// TIA Portal project "color based pick and place" (V16)
// Vorlageprojekt für das Buch mit Zielsystem S7-1200

(* hardware
DEVICE "S7-1200-Station_1"  S7-1200 Station
   slot 0: "Baugruppenträger_0"  Rack  V1.0
   slot 1: "PLC_1"  CPU 1211C DC/DC/DC  6ES7 211-1AE40-0XB0  V4.1
*)

// ===== PLC "PLC_1"  CPU 1211C DC/DC/DC =====

VAR_GLOBAL   // PLC tag table "Standard-Variablentabelle"
   "start" AT %I0.0 : Bool;
   "diffus1" AT %I0.1 : Bool;
   "vision sens" AT %I0.2 : Bool;
   "diffus2" AT %I0.3 : Bool;
   "diffuse3" AT %I0.4 : Bool;
   "emitt1" AT %Q0.0 : Bool;
   "emitt2" AT %Q0.1 : Bool;
   "emitt3" AT %Q0.2 : Bool;
   "conv1" AT %Q0.3 : Bool;
   "conv2" AT %Q0.4 : Bool;
   "conv3" AT %Q0.5 : Bool;
   "diffues2 memory" AT %M0.3 : Bool;
   "diffues3 memory" AT %M0.4 : Bool;
   "diffues1 memory" AT %M0.1 : Bool;
   "vision sensor memory" AT %M0.2 : Bool;
   "z down" AT %Q0.6 : Bool;
   "z sensor(1)" AT %I0.7 : Bool;
   "z snsor  memory" AT %M50.7 : Bool;
   "box detect(1)" AT %I1.0 : Bool;
   "box detect memo" AT %M16.0 : Bool;
   "grab" AT %Q0.7 : Bool;
   "x move" AT %Q1.0 : Bool;
   "x move sens" AT %I1.1 : Bool;
   "x sens mem" AT %M16.1 : Bool;
   "turn left" AT %Q1.1 : Bool;
   "turn right" AT %Q1.2 : Bool;
   "turn sensor" AT %I1.2 : Bool;
   "ton set" AT %M0.5 : Bool;
   "arrive" AT %M0.6 : Bool;
   "retrain" AT %M16.2 : Bool;
   "Tag_1" AT %M16.3 : Bool;
   "Tag_2" AT %M3.0 : Bool;
   "Tag_3" AT %M3.1 : Bool;
   "Tag_4" AT %M3.2 : Bool;
   "reset" AT %M120.0 : Bool;
   "counter reset" AT %I1.3 : Bool;
   "warning light" AT %Q1.3 : Bool;
   "Tag_5" AT %M3.4 : Bool;
   "Tag_6" AT %M10.0 : Bool;
   "Tag_7" AT %M10.1 : Bool;
   "Tag_8" AT %M10.4 : Bool;
   "System_Byte" AT %MB1 : Byte;
   "FirstScan" AT %M1.0 : Bool;
   "DiagStatusUpdate" AT %M1.1 : Bool;
   "AlwaysTRUE" AT %M1.2 : Bool;
   "AlwaysFALSE" AT %M1.3 : Bool;
   "Clock_Byte" AT %MB15 : Byte;
   "Clock_10Hz" AT %M15.0 : Bool;
   "Clock_5Hz" AT %M15.1 : Bool;
   "Clock_2.5Hz" AT %M15.2 : Bool;
   "Clock_2Hz" AT %M15.3 : Bool;
   "Clock_1.25Hz" AT %M15.4 : Bool;
   "Clock_1Hz" AT %M15.5 : Bool;
   "Clock_0.625Hz" AT %M15.6 : Bool;
   "Clock_0.5Hz" AT %M15.7 : Bool;
   "Tag_9" AT %M10.7 : Bool;
   "Tag_10" AT %M50.0 : Bool;
   "Tag_11" AT %M10.2 : Bool;
   "Tag_12" AT %M50.5 : Bool;
   "color not detect latch" AT %M60.0 : Bool;
   "color detect latch" AT %M60.1 : Bool;
   "Tag_13" AT %M70.0 : Bool;
   "turn right reset" AT %M90.0 : Bool;
   "Tag_14" AT %M60.6 : Bool;
   "Tag_15" AT %M100.0 : Bool;
   "Tag_16" AT %M100.1 : Bool;
   "Tag_17" AT %M600.0 : Bool;
   "Tag_18" AT %M600.1 : Bool;
   "Tag_19" AT %M300.3 : Bool;
   "Tag_20" AT %M300.4 : Bool;
   "Tag_21" AT %M700.0 : Bool;
   "Tag_22" AT %M700.1 : Bool;
END_VAR

// folder: System blocks/Program resources

DATA_BLOCK "IEC_Timer_0_DB"   // DB1
{ S7_Optimized_Access := 'TRUE' }
AUTHOR : Simatic
FAMILY : IEC
NAME : IEC_TMR
VERSION : 1.0
// stored: InstanceOfName IEC_TIMER
"IEC_TIMER"
BEGIN
END_DATA_BLOCK

DATA_BLOCK "IEC_Timer_0_DB_1"   // DB2
{ S7_Optimized_Access := 'TRUE' }
AUTHOR : Simatic
FAMILY : IEC
NAME : IEC_TMR
VERSION : 1.0
// stored: InstanceOfName IEC_TIMER
"IEC_TIMER"
BEGIN
END_DATA_BLOCK

DATA_BLOCK "IEC_Counter_0_DB"   // DB3
{ S7_Optimized_Access := 'TRUE' }
AUTHOR : Simatic
FAMILY : IEC
NAME : CNTR
VERSION : 1.0
// stored: InstanceOfName IEC_COUNTER
"IEC_COUNTER"
BEGIN
END_DATA_BLOCK

DATA_BLOCK "IEC_Timer_0_DB_3"   // DB4
{ S7_Optimized_Access := 'TRUE' }
AUTHOR : Simatic
FAMILY : IEC
NAME : IEC_TMR
VERSION : 1.0
// stored: InstanceOfName IEC_TIMER
"IEC_TIMER"
BEGIN
END_DATA_BLOCK

DATA_BLOCK "IEC_Timer_0_DB_2"   // DB5
{ S7_Optimized_Access := 'TRUE' }
AUTHOR : Simatic
FAMILY : IEC
NAME : IEC_TMR
VERSION : 1.0
// stored: InstanceOfName IEC_TIMER
"IEC_TIMER"
BEGIN
END_DATA_BLOCK

DATA_BLOCK "IEC_Counter_1_DB"   // DB6
{ S7_Optimized_Access := 'TRUE' }
AUTHOR : Simatic
FAMILY : IEC
NAME : CNTR
VERSION : 1.0
// stored: InstanceOfName IEC_COUNTER
"IEC_COUNTER"
BEGIN
END_DATA_BLOCK

DATA_BLOCK "IEC_Timer_0_DB_4"   // DB7
{ S7_Optimized_Access := 'TRUE' }
AUTHOR : Simatic
FAMILY : IEC
NAME : IEC_TMR
VERSION : 1.0
// stored: InstanceOfName IEC_TIMER
"IEC_TIMER"
BEGIN
END_DATA_BLOCK

DATA_BLOCK "IEC_Timer_0_DB_5"   // DB8
{ S7_Optimized_Access := 'TRUE' }
AUTHOR : Simatic
FAMILY : IEC
NAME : IEC_TMR
VERSION : 1.0
// stored: InstanceOfName IEC_TIMER
"IEC_TIMER"
BEGIN
END_DATA_BLOCK

// folder: (top level)

FUNCTION "color detect" : Void   // FC1, LAD
{ S7_Optimized_Access := 'TRUE' }
VERSION : 0.1
   VAR_TEMP   // added for the SCL form of the ladder/FBD networks
      _w1 : Bool;
      _w2 : Bool;
      _w3 : Bool;
   END_VAR
BEGIN

REGION Network 1
   // color detect
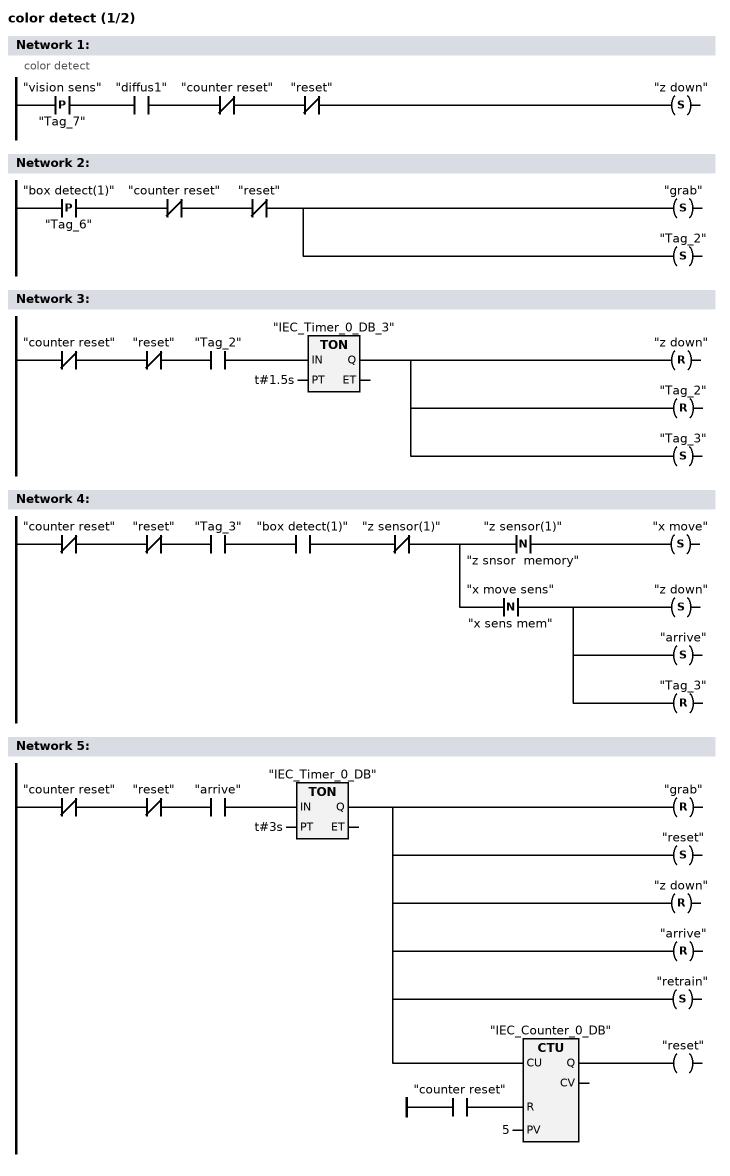
   RUNG wire#powerrail
      P_Contact(operand := "vision sens", bit := "Tag_7")
      Contact( "diffus1" )
      I_Contact( "counter reset" )
      I_Contact( "reset" )
      S_Coil( "z down" )
   END_RUNG
   // the same network as SCL:
   #_w1 := "vision sens" AND NOT "Tag_7";   // rising edge of "vision sens"
   "Tag_7" := "vision sens";
   IF #_w1 AND "diffus1" AND NOT "counter reset" AND NOT "reset" THEN "z down" := TRUE; END_IF;
END_REGION

REGION Network 2
   RUNG wire#powerrail
      P_Contact(operand := "box detect(1)", bit := "Tag_6")
      I_Contact( "counter reset" )
      I_Contact( "reset" )
      wire#w1
      S_Coil( "grab" )
   END_RUNG
   RUNG wire#w1
      S_Coil( "Tag_2" )
   END_RUNG
   // the same network as SCL:
   #_w1 := "box detect(1)" AND NOT "Tag_6";   // rising edge of "box detect(1)"
   "Tag_6" := "box detect(1)";
   IF #_w1 AND NOT "counter reset" AND NOT "reset" THEN
       "grab" := TRUE;
       "Tag_2" := TRUE;
   END_IF;
END_REGION

REGION Network 3
   "IEC_Timer_0_DB_3".TON(IN := NOT "counter reset" AND NOT "reset" AND "Tag_2", PT := t#1.5s);
   IF "IEC_Timer_0_DB_3".Q THEN
       "z down" := FALSE;
       "Tag_2" := FALSE;
       "Tag_3" := TRUE;
   END_IF;
END_REGION

REGION Network 4
   RUNG wire#powerrail
      I_Contact( "counter reset" )
      I_Contact( "reset" )
      Contact( "Tag_3" )
      Contact( "box detect(1)" )
      I_Contact( "z sensor(1)" )
      wire#w1
      N_Contact(operand := "z sensor(1)", bit := "z snsor  memory")
      S_Coil( "x move" )
   END_RUNG
   RUNG wire#w1
      N_Contact(operand := "x move sens", bit := "x sens mem")
      wire#w2
      S_Coil( "z down" )
   END_RUNG
   RUNG wire#w2
      S_Coil( "arrive" )
   END_RUNG
   RUNG wire#w2
      R_Coil( "Tag_3" )
   END_RUNG
   // the same network as SCL:
   #_w1 := NOT "counter reset" AND NOT "reset" AND "Tag_3" AND "box detect(1)" AND NOT "z sensor(1)";
   #_w2 := #_w1 AND NOT "z sensor(1)" AND "z snsor  memory";   // falling edge of "z sensor(1)"
   "z snsor  memory" := "z sensor(1)";
   IF #_w2 THEN "x move" := TRUE; END_IF;
   #_w3 := #_w1 AND NOT "x move sens" AND "x sens mem";   // falling edge of "x move sens"
   "x sens mem" := "x move sens";
   IF #_w3 THEN
       "z down" := TRUE;
       "arrive" := TRUE;
       "Tag_3" := FALSE;
   END_IF;
END_REGION

REGION Network 5
   "IEC_Timer_0_DB".TON(IN := NOT "counter reset" AND NOT "reset" AND "arrive", PT := t#3s);
   IF "IEC_Timer_0_DB".Q THEN
       "grab" := FALSE;
       "reset" := TRUE;
       "z down" := FALSE;
       "arrive" := FALSE;
       "retrain" := TRUE;
   END_IF;
   "IEC_Counter_0_DB".CTU(CU := "IEC_Timer_0_DB".Q, R := "counter reset", PV := 5);
   "reset" := "IEC_Counter_0_DB".Q;
END_REGION

REGION Network 6
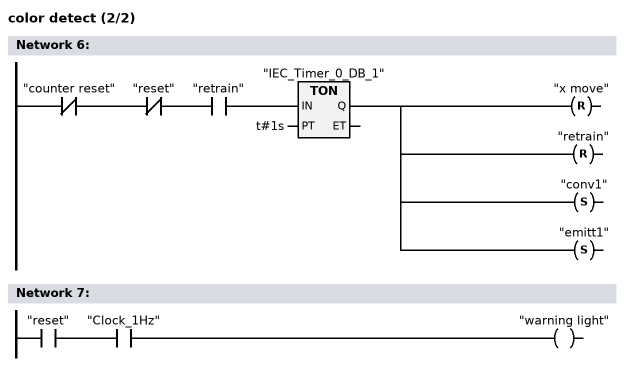
   "IEC_Timer_0_DB_1".TON(IN := NOT "counter reset" AND NOT "reset" AND "retrain", PT := t#1s);
   IF "IEC_Timer_0_DB_1".Q THEN
       "x move" := FALSE;
       "retrain" := FALSE;
       "conv1" := TRUE;
       "emitt1" := TRUE;
   END_IF;
END_REGION

REGION Network 7
   RUNG wire#powerrail
      Contact( "reset" )
      Contact( "Clock_1Hz" )
      Coil( "warning light" )
   END_RUNG
   // the same network as SCL:
   "warning light" := "reset" AND "Clock_1Hz";
END_REGION
END_FUNCTION

FUNCTION "color not detect" : Void   // FC2, LAD
{ S7_Optimized_Access := 'TRUE' }
VERSION : 0.1
   VAR_TEMP   // added for the SCL form of the ladder/FBD networks
      _w1 : Bool;
      _w2 : Bool;
      _w3 : Bool;
      _w4 : Bool;
   END_VAR
BEGIN

REGION Network 1
   // color detect
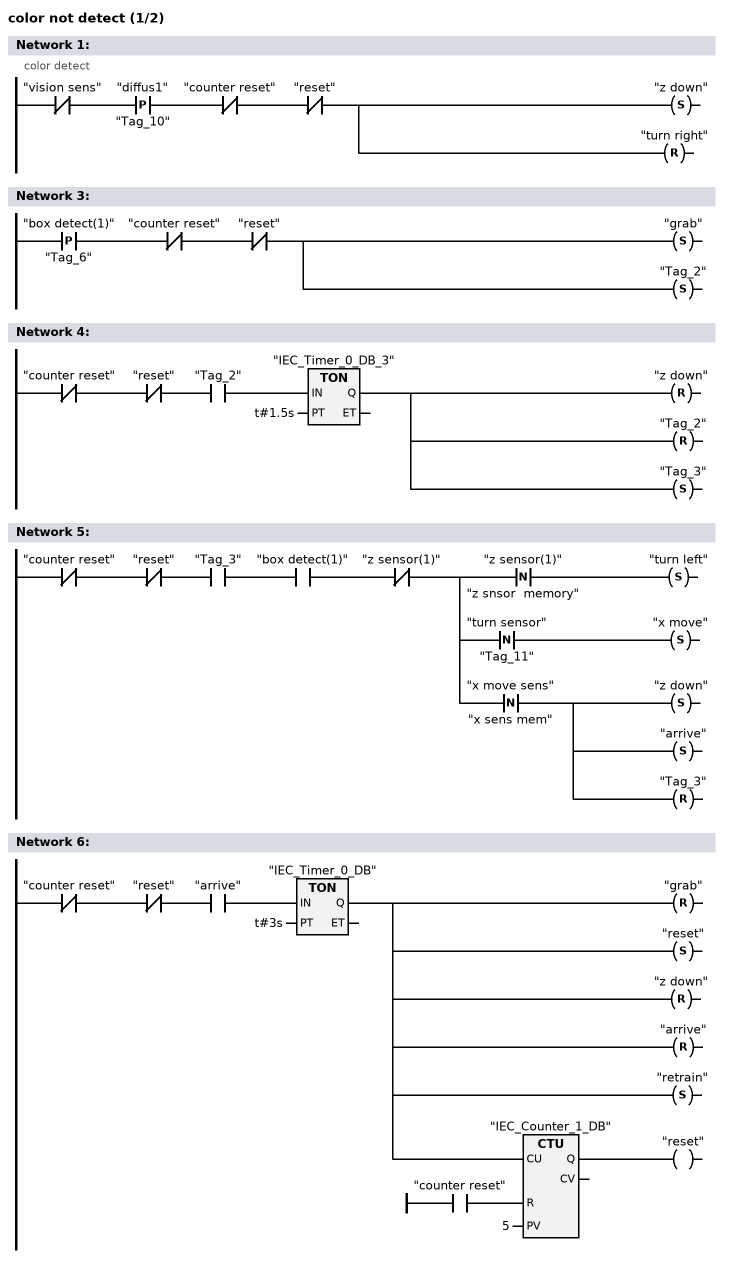
   RUNG wire#powerrail
      I_Contact( "vision sens" )
      P_Contact(operand := "diffus1", bit := "Tag_10")
      I_Contact( "counter reset" )
      I_Contact( "reset" )
      wire#w1
      S_Coil( "z down" )
   END_RUNG
   RUNG wire#w1
      R_Coil( "turn right" )
   END_RUNG
   // the same network as SCL:
   #_w1 := NOT "vision sens" AND "diffus1" AND NOT "Tag_10";   // rising edge of "diffus1"
   "Tag_10" := "diffus1";
   IF #_w1 AND NOT "counter reset" AND NOT "reset" THEN
       "z down" := TRUE;
       "turn right" := FALSE;
   END_IF;
END_REGION

REGION Network 3
   RUNG wire#powerrail
      P_Contact(operand := "box detect(1)", bit := "Tag_6")
      I_Contact( "counter reset" )
      I_Contact( "reset" )
      wire#w1
      S_Coil( "grab" )
   END_RUNG
   RUNG wire#w1
      S_Coil( "Tag_2" )
   END_RUNG
   // the same network as SCL:
   #_w1 := "box detect(1)" AND NOT "Tag_6";   // rising edge of "box detect(1)"
   "Tag_6" := "box detect(1)";
   IF #_w1 AND NOT "counter reset" AND NOT "reset" THEN
       "grab" := TRUE;
       "Tag_2" := TRUE;
   END_IF;
END_REGION

REGION Network 4
   "IEC_Timer_0_DB_3".TON(IN := NOT "counter reset" AND NOT "reset" AND "Tag_2", PT := t#1.5s);
   IF "IEC_Timer_0_DB_3".Q THEN
       "z down" := FALSE;
       "Tag_2" := FALSE;
       "Tag_3" := TRUE;
   END_IF;
END_REGION

REGION Network 5
   RUNG wire#powerrail
      I_Contact( "counter reset" )
      I_Contact( "reset" )
      Contact( "Tag_3" )
      Contact( "box detect(1)" )
      I_Contact( "z sensor(1)" )
      wire#w1
      N_Contact(operand := "z sensor(1)", bit := "z snsor  memory")
      S_Coil( "turn left" )
   END_RUNG
   RUNG wire#w1
      N_Contact(operand := "turn sensor", bit := "Tag_11")
      S_Coil( "x move" )
   END_RUNG
   RUNG wire#w1
      N_Contact(operand := "x move sens", bit := "x sens mem")
      wire#w2
      S_Coil( "z down" )
   END_RUNG
   RUNG wire#w2
      S_Coil( "arrive" )
   END_RUNG
   RUNG wire#w2
      R_Coil( "Tag_3" )
   END_RUNG
   // the same network as SCL:
   #_w1 := NOT "counter reset" AND NOT "reset" AND "Tag_3" AND "box detect(1)" AND NOT "z sensor(1)";
   #_w2 := #_w1 AND NOT "z sensor(1)" AND "z snsor  memory";   // falling edge of "z sensor(1)"
   "z snsor  memory" := "z sensor(1)";
   IF #_w2 THEN "turn left" := TRUE; END_IF;
   #_w3 := #_w1 AND NOT "turn sensor" AND "Tag_11";   // falling edge of "turn sensor"
   "Tag_11" := "turn sensor";
   IF #_w3 THEN "x move" := TRUE; END_IF;
   #_w4 := #_w1 AND NOT "x move sens" AND "x sens mem";   // falling edge of "x move sens"
   "x sens mem" := "x move sens";
   IF #_w4 THEN
       "z down" := TRUE;
       "arrive" := TRUE;
       "Tag_3" := FALSE;
   END_IF;
END_REGION

REGION Network 6
   "IEC_Timer_0_DB".TON(IN := NOT "counter reset" AND NOT "reset" AND "arrive", PT := t#3s);
   IF "IEC_Timer_0_DB".Q THEN
       "grab" := FALSE;
       "reset" := TRUE;
       "z down" := FALSE;
       "arrive" := FALSE;
       "retrain" := TRUE;
   END_IF;
   "IEC_Counter_1_DB".CTU(CU := "IEC_Timer_0_DB".Q, R := "counter reset", PV := 5);
   "reset" := "IEC_Counter_1_DB".Q;
END_REGION

REGION Network 7
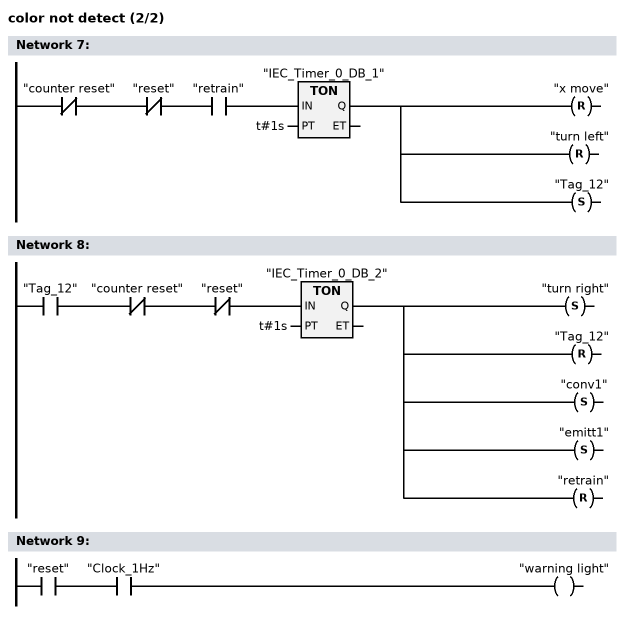
   "IEC_Timer_0_DB_1".TON(IN := NOT "counter reset" AND NOT "reset" AND "retrain", PT := t#1s);
   IF "IEC_Timer_0_DB_1".Q THEN
       "x move" := FALSE;
       "turn left" := FALSE;
       "Tag_12" := TRUE;
   END_IF;
END_REGION

REGION Network 8
   "IEC_Timer_0_DB_2".TON(IN := "Tag_12" AND NOT "counter reset" AND NOT "reset", PT := t#1s);
   IF "IEC_Timer_0_DB_2".Q THEN
       "turn right" := TRUE;
       "Tag_12" := FALSE;
       "conv1" := TRUE;
       "emitt1" := TRUE;
       "retrain" := FALSE;
   END_IF;
END_REGION

REGION Network 9
   RUNG wire#powerrail
      Contact( "reset" )
      Contact( "Clock_1Hz" )
      Coil( "warning light" )
   END_RUNG
   // the same network as SCL:
   "warning light" := "reset" AND "Clock_1Hz";
END_REGION
END_FUNCTION

FUNCTION "MHJ-PLC-Lab-Function-S71200" : Void   // FC9000, SCL
{ S7_Optimized_Access := 'TRUE' }
VERSION : 0.1
   VAR_TEMP
      rdTimeReturn : Int;
      outputTime : DTL;
      SyncVal : Byte;
      forVal : Int;
      forVal_2 : Int;
      Value : Byte;
   END_VAR
   VAR CONSTANT
      CompVal : Byte := 16#34;
      Value_01 : Byte := 16#11;
      Value_01_DW : DWord := 16#A165_D992;
      Value_02_DW : DWord := 16#58BE_4401;
   END_VAR
BEGIN

   #Value:=PEEK(area := 16#82,
        dbNumber := 0,
        byteOffset := 511);
   #Value := #Value + 1;

   POKE(area := 16#82,
        dbNumber := 0,
        byteOffset := 511,
        value := #Value);

   POKE(area:=16#81,
        dbNumber:=0,
        byteOffset:=1016,
        value:=#Value_01_DW);
   POKE(area := 16#81,
        dbNumber := 0,
        byteOffset := 1020,
        value := #Value_02_DW);

   POKE(area := 16#81,
        dbNumber := 0,
        byteOffset := 511,
        value := B#16#00);

   FOR #forVal := 0 TO 120 DO
       FOR #forVal_2:=0 TO 10 DO
           #rdTimeReturn:=RD_SYS_T(#outputTime);
           #rdTimeReturn := WR_SYS_T(#outputTime);
           #rdTimeReturn := RD_SYS_T(#outputTime);
           #rdTimeReturn := WR_SYS_T(#outputTime);
       END_FOR;
       #SyncVal:= PEEK(area := 16#81,
                      dbNumber := 0,
                      byteOffset := 511);
       IF #SyncVal = #CompVal THEN
          GOTO M_1;
       END_IF;
   END_FOR;
   RETURN;

   M_1:
   POKE(area := 16#81,
        dbNumber := 0,
        byteOffset := 511,
        value := B#16#0);
END_FUNCTION

ORGANIZATION_BLOCK "Main"   // OB1, LAD, ProgramCycle
TITLE = "Main Program Sweep (Cycle)"
{ S7_Optimized_Access := 'TRUE' }
VERSION : 0.1
   VAR_INPUT
      Initial_Call : Bool;   // Initial call of this OB
      Remanence : Bool;   // =True, if remanent data are available
   END_VAR
   VAR_TEMP   // added for the SCL form of the ladder/FBD networks
      _w1 : Bool;
      _w2 : Bool;
      _w3 : Bool;
      _w4 : Bool;
   END_VAR
BEGIN

REGION Network 1
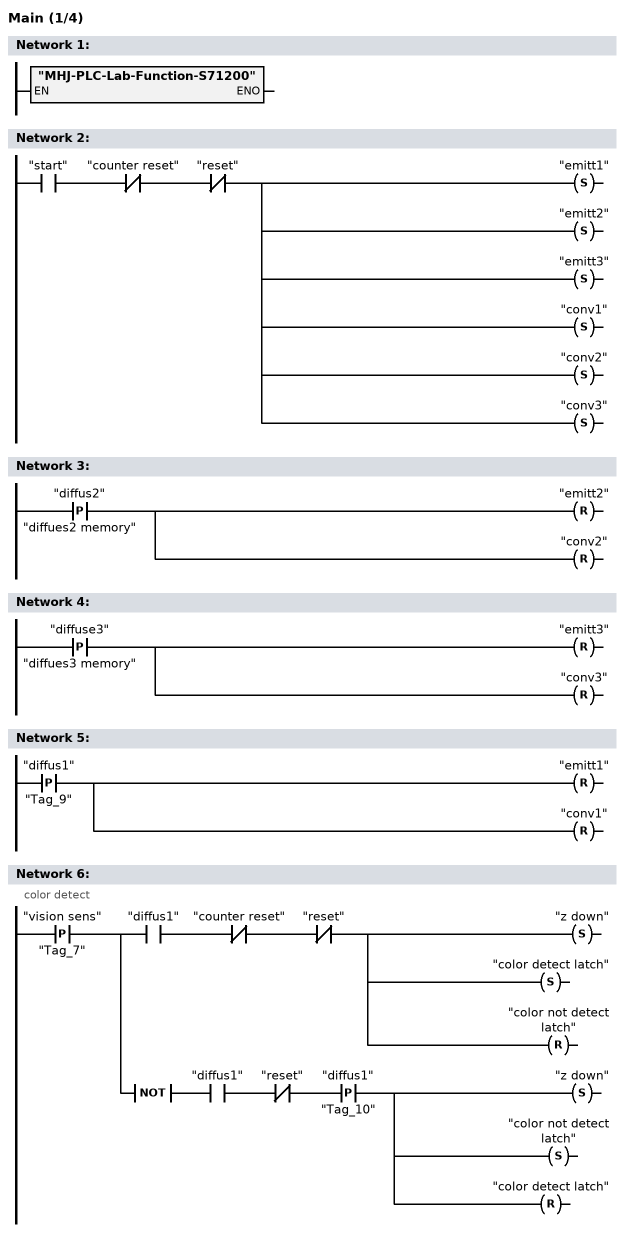
   RUNG wire#powerrail
      "MHJ-PLC-Lab-Function-S71200"()
   END_RUNG
   // the same network as SCL:
   "MHJ-PLC-Lab-Function-S71200"();
END_REGION

REGION Network 2
   RUNG wire#powerrail
      Contact( "start" )
      I_Contact( "counter reset" )
      I_Contact( "reset" )
      wire#w1
      S_Coil( "emitt1" )
   END_RUNG
   RUNG wire#w1
      S_Coil( "emitt2" )
   END_RUNG
   RUNG wire#w1
      S_Coil( "emitt3" )
   END_RUNG
   RUNG wire#w1
      S_Coil( "conv1" )
   END_RUNG
   RUNG wire#w1
      S_Coil( "conv2" )
   END_RUNG
   RUNG wire#w1
      S_Coil( "conv3" )
   END_RUNG
   // the same network as SCL:
   IF "start" AND NOT "counter reset" AND NOT "reset" THEN
       "emitt1" := TRUE;
       "emitt2" := TRUE;
       "emitt3" := TRUE;
       "conv1" := TRUE;
       "conv2" := TRUE;
       "conv3" := TRUE;
   END_IF;
END_REGION

REGION Network 3
   RUNG wire#powerrail
      P_Contact(operand := "diffus2", bit := "diffues2 memory")
      wire#w1
      R_Coil( "emitt2" )
   END_RUNG
   RUNG wire#w1
      R_Coil( "conv2" )
   END_RUNG
   // the same network as SCL:
   #_w1 := "diffus2" AND NOT "diffues2 memory";   // rising edge of "diffus2"
   "diffues2 memory" := "diffus2";
   IF #_w1 THEN
       "emitt2" := FALSE;
       "conv2" := FALSE;
   END_IF;
END_REGION

REGION Network 4
   RUNG wire#powerrail
      P_Contact(operand := "diffuse3", bit := "diffues3 memory")
      wire#w1
      R_Coil( "emitt3" )
   END_RUNG
   RUNG wire#w1
      R_Coil( "conv3" )
   END_RUNG
   // the same network as SCL:
   #_w1 := "diffuse3" AND NOT "diffues3 memory";   // rising edge of "diffuse3"
   "diffues3 memory" := "diffuse3";
   IF #_w1 THEN
       "emitt3" := FALSE;
       "conv3" := FALSE;
   END_IF;
END_REGION

REGION Network 5
   RUNG wire#powerrail
      P_Contact(operand := "diffus1", bit := "Tag_9")
      wire#w1
      R_Coil( "emitt1" )
   END_RUNG
   RUNG wire#w1
      R_Coil( "conv1" )
   END_RUNG
   // the same network as SCL:
   #_w1 := "diffus1" AND NOT "Tag_9";   // rising edge of "diffus1"
   "Tag_9" := "diffus1";
   IF #_w1 THEN
       "emitt1" := FALSE;
       "conv1" := FALSE;
   END_IF;
END_REGION

REGION Network 6
   // color detect
   RUNG wire#powerrail
      P_Contact(operand := "vision sens", bit := "Tag_7")
      wire#w1
      Contact( "diffus1" )
      I_Contact( "counter reset" )
      I_Contact( "reset" )
      wire#w2
      S_Coil( "z down" )
   END_RUNG
   RUNG wire#w2
      S_Coil( "color detect latch" )
   END_RUNG
   RUNG wire#w2
      R_Coil( "color not detect latch" )
   END_RUNG
   RUNG wire#w1
      Not()
      Contact( "diffus1" )
      I_Contact( "reset" )
      P_Contact(operand := "diffus1", bit := "Tag_10")
      wire#w3
      S_Coil( "z down" )
   END_RUNG
   RUNG wire#w3
      S_Coil( "color not detect latch" )
   END_RUNG
   RUNG wire#w3
      R_Coil( "color detect latch" )
   END_RUNG
   // the same network as SCL:
   #_w1 := "vision sens" AND NOT "Tag_7";   // rising edge of "vision sens"
   "Tag_7" := "vision sens";
   IF #_w1 AND "diffus1" AND NOT "counter reset" AND NOT "reset" THEN
       "z down" := TRUE;
       "color detect latch" := TRUE;
       "color not detect latch" := FALSE;
   END_IF;
   #_w2 := NOT #_w1 AND "diffus1" AND NOT "reset" AND "diffus1" AND NOT "Tag_10";   // rising edge of "diffus1"
   "Tag_10" := "diffus1";
   IF #_w2 THEN
       "z down" := TRUE;
       "color not detect latch" := TRUE;
       "color detect latch" := FALSE;
   END_IF;
END_REGION

REGION Network 7
   // common item grab
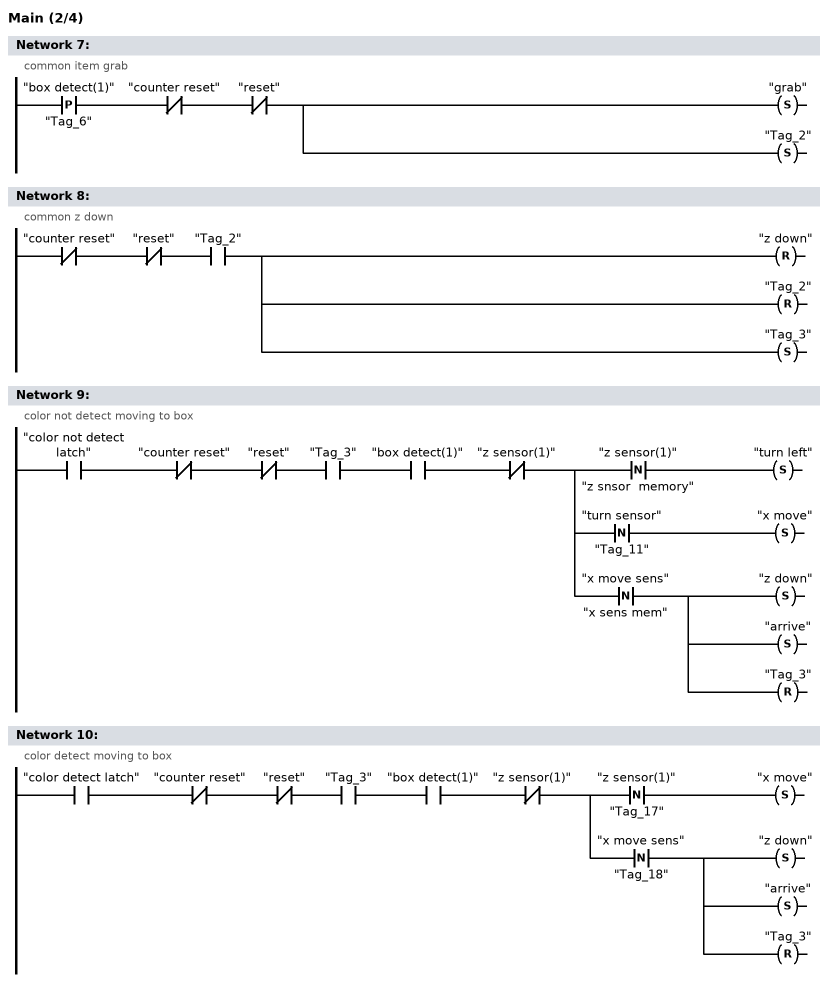
   RUNG wire#powerrail
      P_Contact(operand := "box detect(1)", bit := "Tag_6")
      I_Contact( "counter reset" )
      I_Contact( "reset" )
      wire#w1
      S_Coil( "grab" )
   END_RUNG
   RUNG wire#w1
      S_Coil( "Tag_2" )
   END_RUNG
   // the same network as SCL:
   #_w1 := "box detect(1)" AND NOT "Tag_6";   // rising edge of "box detect(1)"
   "Tag_6" := "box detect(1)";
   IF #_w1 AND NOT "counter reset" AND NOT "reset" THEN
       "grab" := TRUE;
       "Tag_2" := TRUE;
   END_IF;
END_REGION

REGION Network 8
   // common z down
   RUNG wire#powerrail
      I_Contact( "counter reset" )
      I_Contact( "reset" )
      Contact( "Tag_2" )
      wire#w1
      R_Coil( "z down" )
   END_RUNG
   RUNG wire#w1
      R_Coil( "Tag_2" )
   END_RUNG
   RUNG wire#w1
      S_Coil( "Tag_3" )
   END_RUNG
   // the same network as SCL:
   IF NOT "counter reset" AND NOT "reset" AND "Tag_2" THEN "z down" := FALSE; END_IF;
   #_w1 := NOT "counter reset" AND NOT "reset" AND "Tag_2";
   IF #_w1 THEN
       "Tag_2" := FALSE;
       "Tag_3" := TRUE;
   END_IF;
END_REGION

REGION Network 9
   // color not detect moving to box
   RUNG wire#powerrail
      Contact( "color not detect latch" )
      I_Contact( "counter reset" )
      I_Contact( "reset" )
      Contact( "Tag_3" )
      Contact( "box detect(1)" )
      I_Contact( "z sensor(1)" )
      wire#w1
      N_Contact(operand := "z sensor(1)", bit := "z snsor  memory")
      S_Coil( "turn left" )
   END_RUNG
   RUNG wire#w1
      N_Contact(operand := "turn sensor", bit := "Tag_11")
      S_Coil( "x move" )
   END_RUNG
   RUNG wire#w1
      N_Contact(operand := "x move sens", bit := "x sens mem")
      wire#w2
      S_Coil( "z down" )
   END_RUNG
   RUNG wire#w2
      S_Coil( "arrive" )
   END_RUNG
   RUNG wire#w2
      R_Coil( "Tag_3" )
   END_RUNG
   // the same network as SCL:
   #_w1 := "color not detect latch" AND NOT "counter reset" AND NOT "reset" AND "Tag_3" AND "box detect(1)" AND NOT "z sensor(1)";
   #_w2 := #_w1 AND NOT "z sensor(1)" AND "z snsor  memory";   // falling edge of "z sensor(1)"
   "z snsor  memory" := "z sensor(1)";
   IF #_w2 THEN "turn left" := TRUE; END_IF;
   #_w3 := #_w1 AND NOT "turn sensor" AND "Tag_11";   // falling edge of "turn sensor"
   "Tag_11" := "turn sensor";
   IF #_w3 THEN "x move" := TRUE; END_IF;
   #_w4 := #_w1 AND NOT "x move sens" AND "x sens mem";   // falling edge of "x move sens"
   "x sens mem" := "x move sens";
   IF #_w4 THEN
       "z down" := TRUE;
       "arrive" := TRUE;
       "Tag_3" := FALSE;
   END_IF;
END_REGION

REGION Network 10
   // color detect moving to box
   RUNG wire#powerrail
      Contact( "color detect latch" )
      I_Contact( "counter reset" )
      I_Contact( "reset" )
      Contact( "Tag_3" )
      Contact( "box detect(1)" )
      I_Contact( "z sensor(1)" )
      wire#w1
      N_Contact(operand := "z sensor(1)", bit := "Tag_17")
      S_Coil( "x move" )
   END_RUNG
   RUNG wire#w1
      N_Contact(operand := "x move sens", bit := "Tag_18")
      wire#w2
      S_Coil( "z down" )
   END_RUNG
   RUNG wire#w2
      S_Coil( "arrive" )
   END_RUNG
   RUNG wire#w2
      R_Coil( "Tag_3" )
   END_RUNG
   // the same network as SCL:
   #_w1 := "color detect latch" AND NOT "counter reset" AND NOT "reset" AND "Tag_3" AND "box detect(1)" AND NOT "z sensor(1)";
   #_w2 := #_w1 AND NOT "z sensor(1)" AND "Tag_17";   // falling edge of "z sensor(1)"
   "Tag_17" := "z sensor(1)";
   IF #_w2 THEN "x move" := TRUE; END_IF;
   #_w3 := #_w1 AND NOT "x move sens" AND "Tag_18";   // falling edge of "x move sens"
   "Tag_18" := "x move sens";
   IF #_w3 THEN
       "z down" := TRUE;
       "arrive" := TRUE;
       "Tag_3" := FALSE;
   END_IF;
END_REGION

REGION Network 11
   // common arrive to box
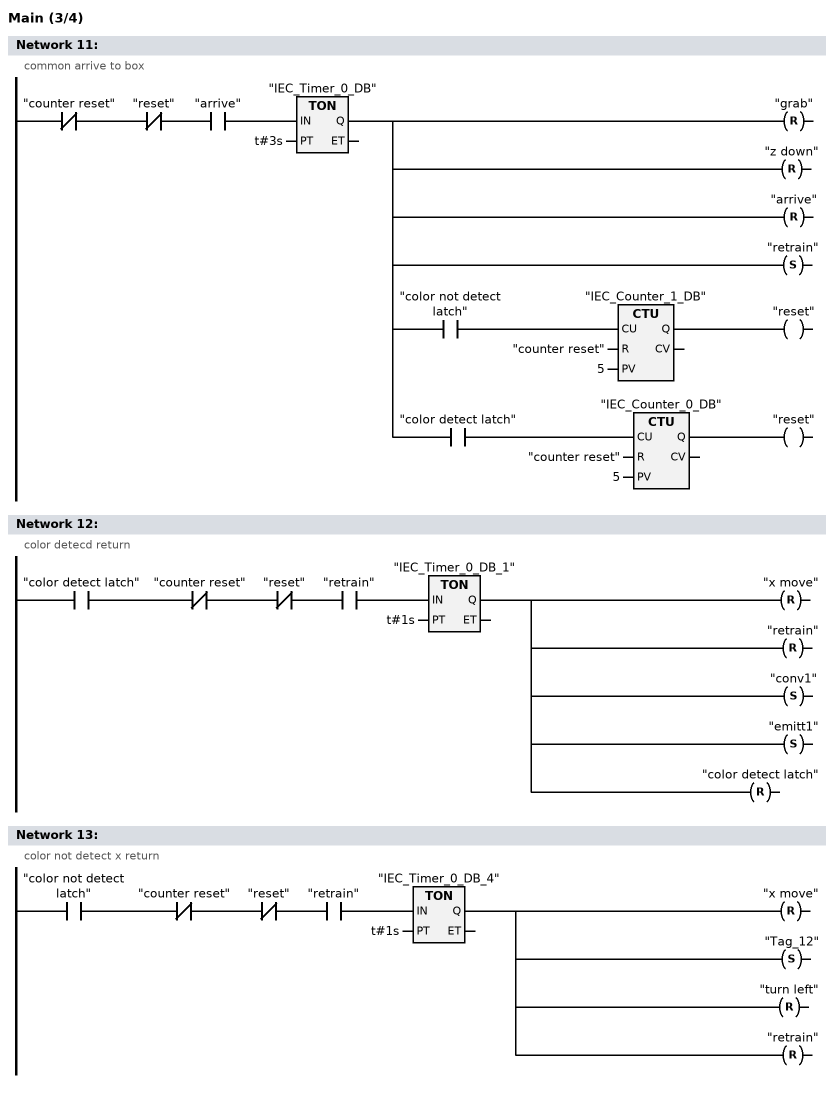
   "IEC_Timer_0_DB".TON(IN := NOT "counter reset" AND NOT "reset" AND "arrive", PT := t#3s);
   IF "IEC_Timer_0_DB".Q THEN
       "grab" := FALSE;
       "z down" := FALSE;
       "arrive" := FALSE;
       "retrain" := TRUE;
   END_IF;
   "IEC_Counter_1_DB".CTU(CU := "IEC_Timer_0_DB".Q AND "color not detect latch", R := "counter reset", PV := 5);
   "reset" := "IEC_Counter_1_DB".Q;
   "IEC_Counter_0_DB".CTU(CU := "IEC_Timer_0_DB".Q AND "color detect latch", R := "counter reset", PV := 5);
   "reset" := "IEC_Counter_0_DB".Q;
END_REGION

REGION Network 12
   // color detecd return
   "IEC_Timer_0_DB_1".TON(IN := "color detect latch" AND NOT "counter reset" AND NOT "reset" AND "retrain",
                          PT := t#1s);
   IF "IEC_Timer_0_DB_1".Q THEN
       "x move" := FALSE;
       "retrain" := FALSE;
       "conv1" := TRUE;
       "emitt1" := TRUE;
       "color detect latch" := FALSE;
   END_IF;
END_REGION

REGION Network 13
   // color not detect x return
   "IEC_Timer_0_DB_4".TON(IN := "color not detect latch" AND NOT "counter reset" AND NOT "reset" AND "retrain",
                          PT := t#1s);
   IF "IEC_Timer_0_DB_4".Q THEN
       "x move" := FALSE;
       "Tag_12" := TRUE;
       "turn left" := FALSE;
       "retrain" := FALSE;
   END_IF;
END_REGION

REGION Network 14
   // color not detect
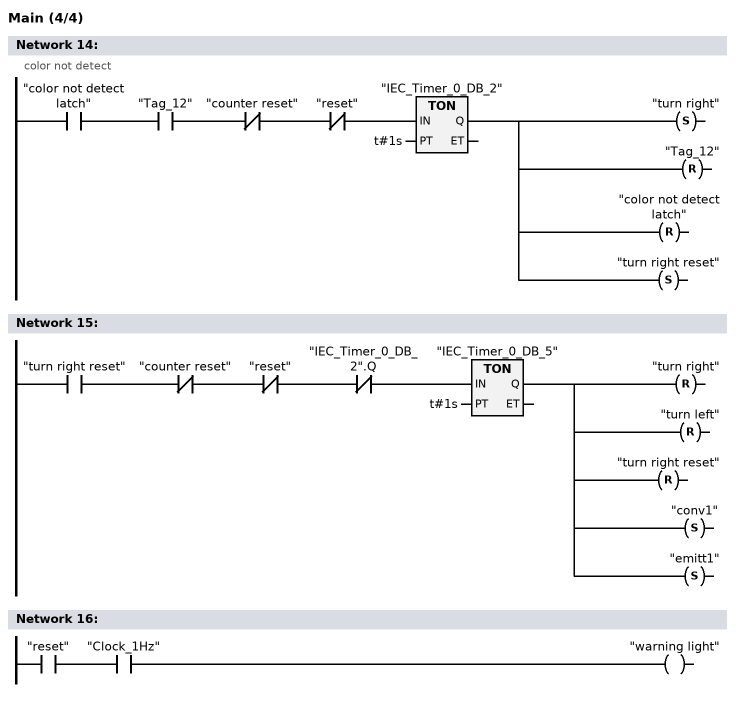
   "IEC_Timer_0_DB_2".TON(IN := "color not detect latch" AND "Tag_12" AND NOT "counter reset" AND NOT "reset",
                          PT := t#1s);
   IF "IEC_Timer_0_DB_2".Q THEN
       "turn right" := TRUE;
       "Tag_12" := FALSE;
       "color not detect latch" := FALSE;
       "turn right reset" := TRUE;
   END_IF;
END_REGION

REGION Network 15
   "IEC_Timer_0_DB_5".TON(IN := "turn right reset" AND NOT "counter reset" AND NOT "reset" AND NOT "IEC_Timer_0_DB_2".Q,
                          PT := t#1s);
   IF "IEC_Timer_0_DB_5".Q THEN
       "turn right" := FALSE;
       "turn left" := FALSE;
       "turn right reset" := FALSE;
       "conv1" := TRUE;
       "emitt1" := TRUE;
   END_IF;
END_REGION

REGION Network 16
   RUNG wire#powerrail
      Contact( "reset" )
      Contact( "Clock_1Hz" )
      Coil( "warning light" )
   END_RUNG
   // the same network as SCL:
   "warning light" := "reset" AND "Clock_1Hz";
END_REGION
END_ORGANIZATION_BLOCK